PROGRAM PRG_ROOTS
VAR
END_VAR

(*EM1L0*)
(*Roots Pump Chamber 1*)
(*gauges*)
GEM1_GPI_60(PG=>);
GEM1_GPI_61(PG=>);
GEM1_GPI_71(PG=>);

(*Isolation Valve*)
GEM1_VRC_60(Pump:=GEM1_PRO_60.q_stPump,Gauge:=GEM1_GPI_60.PG,i_xExtILK_OK:=TRUE);
GEM1_VRC_70(Pump:=GEM1_PRO_70.q_stPump,Gauge:=GEM1_GPI_60.PG,i_xExtILK_OK:=TRUE);


(* dry pump*)
GEM1_PRO_60();
GEM1_PRO_70();




(*EM2L0*)
(*Roots Pump Chamber 1*)
(*gauges*)
GEM2_GPI_10(PG=>);
GEM2_GPI_11(PG=>);
GEM2_GPI_21(PG=>);

(*Isolation Valve*)
GEM2_VRC_10(Pump:=GEM2_PRO_10.q_stPump,Gauge:=GEM2_GPI_10.PG,i_xExtILK_OK:=TRUE);
GEM2_VRC_20(Pump:=GEM2_PRO_20.q_stPump,Gauge:=GEM2_GPI_10.PG,i_xExtILK_OK:=TRUE);

(* dry pump*)
GEM2_PRO_10();
GEM2_PRO_20();

END_PROGRAM

(* stored: Version 1.1.0.1, ProductVersion 3.1.4022.16
   POU PRG_ROOTS: Id {573f7847-bda8-45d7-9541-d46f5c27ae92}, SpecialFunc None *)
